Yaskawa INFORM job: MASTER.JBI

/JOB
//NAME MASTER
//POS
///NPOS 0,0,0,0,0,0
//INST
///DATE 2019/03/13 18:25
///ATTR SC,RW
///GROUP1 RB1
NOP
SFTOF
CLEAR STACK
CALL JOB:RESTORSTION
'RETURN ORIGIN
CALL JOB:HOME-RETURN IF IN#(7)=ON
*HOME
DIN B000 SOUT#(120)
IFTHENEXP B000=1 ANDEXP B001=0
	 JUMP *LOOP
ENDIF
*LOOP
CALL JOB:LOOP-MODEL
JUMP *HOME
END
